# B&R Automation Studio project 8238 (part 12)

#### msgBinSearchHelpTxtLine.st
```iecst
(********************************************************************
 * COPYRIGHT -- Herbert Kannegiesser GmbH
 ********************************************************************
 * Library: KGlibMsg
 * File: msgBinSearchTxtLine.st
 * Author: kuehne
 * Created: November 29, 2011
 ********************************************************************
 * Implementation of library KGlibMsg
 ********************************************************************)

(* TODO: Add your comment here *)
FUNCTION_BLOCK msgBinSearchHelpTxtLine
	wStatus := MNMSG_STAT_NOTFOUND;
	wMsgPos := 65535;
	IF bTupel = 0 OR bTupel > 3 THEN
		RETURN;
	END_IF;
	IF bTupel = 1 THEN
		IF (wFunctionID < 1) OR (wCntMsgHelpTxt < 1) THEN
			RETURN;
		END_IF;
	END_IF;
	IF bTupel = 2 OR bTupel = 3 THEN
		IF (wFunctionID < 1) OR (wNumber < 1) OR (wCntMsgHelpTxt < 1) THEN
			RETURN;
		END_IF;
	END_IF;
	wPosMin := 0;
	wPosBeg := wPosMin;
	wPosEnd := wPosMin + wCntMsgHelpTxt - 1;
	IF wPosEnd = wPosBeg THEN
		CASE bTupel OF
			1:
				IF (MsgHelpTxtList[wPosBeg].wFunctionID = wFunctionID) THEN
					wMsgPos := wPosBeg;
					wStatus := ERR_OK;
					RETURN;
				ELSE
					RETURN;
				END_IF;
			2:
				IF (MsgHelpTxtList[wPosBeg].wFunctionID = wFunctionID) AND (MsgHelpTxtList[wPosBeg].wNumber = wNumber) THEN
					wMsgPos := wPosBeg;
					wStatus := ERR_OK;
					RETURN;
				ELSE
					RETURN;
				END_IF;
			3:
				IF (MsgHelpTxtList[wPosBeg].wFunctionID = wFunctionID) AND (MsgHelpTxtList[wPosBeg].wNumber = wNumber) AND ((MsgHelpTxtList[wPosBeg].wInstance = wInstance) OR (wInstance = 0)) THEN
					wMsgPos := wPosBeg;
					wStatus := ERR_OK;
					RETURN;
				ELSE
					RETURN;
				END_IF;
		END_CASE;
	END_IF;
	wPosMin := 1;
	wPosBeg := wPosMin;
	wPosMax := wPosMin + wCntMsgHelpTxt - 1;
	wPosEnd := wPosMin + wCntMsgHelpTxt - 1;
	wPos := (wPosMin + wPosMax) / 2;
	xPosFound := FALSE;
	WHILE NOT xPosFound DO
		IF ((wPos = (wPosBeg + 1)) OR (wPos = wPosBeg)) AND NOT xPosFound THEN
			wPos := wPosBeg;
			IF (MsgHelpTxtList[wPos].wFunctionID > wFunctionID) AND (MsgHelpTxtList[wPos + 1].wFunctionID > wFunctionID) THEN
				wPos := wPosBeg + 0;
				xPosFound := TRUE;
			ELSIF (MsgHelpTxtList[wPos].wFunctionID < wFunctionID) AND (MsgHelpTxtList[wPos + 1].wFunctionID > wFunctionID) THEN
				wPos := wPosBeg + 1;
				xPosFound := TRUE;
			ELSIF (MsgHelpTxtList[wPos].wFunctionID < wFunctionID) AND (MsgHelpTxtList[wPos + 1].wFunctionID = wFunctionID) THEN
				wPos := wPosBeg + 1;
				xPosFound := TRUE;
			ELSIF (MsgHelpTxtList[wPos].wFunctionID < wFunctionID) AND (MsgHelpTxtList[wPos + 1].wFunctionID < wFunctionID) THEN
				IF wPosEnd = (wPosBeg + 1) THEN
					wCnt := wPosBeg;
					WHILE MsgHelpTxtList[wCnt].wFunctionID < wFunctionID AND (wCnt < wPosEnd) DO
						wCnt := wCnt + 1;
					END_WHILE;
					wPos := wCnt;
				ELSE
					wPos := wPosBeg + 2;
					IF NOT (MsgHelpTxtList[wPos].wFunctionID = wFunctionID) THEN
						wCnt := wPosBeg;
						WHILE MsgHelpTxtList[wCnt].wFunctionID < wFunctionID AND (wCnt < wPosEnd) DO
							wCnt := wCnt + 1;
						END_WHILE;
						wPos := wCnt;
					END_IF;
				END_IF;
				xPosFound := TRUE;
			ELSIF (MsgHelpTxtList[wPos].wFunctionID = wFunctionID) AND (MsgHelpTxtList[wPos + 1].wFunctionID > wFunctionID) THEN
				wPos := wPosBeg + 0;
				xPosFound := TRUE;
			ELSIF (MsgHelpTxtList[wPos].wFunctionID = wFunctionID) AND (MsgHelpTxtList[wPos + 1].wFunctionID = wFunctionID) THEN
				wPos := wPosBeg + 0;
				xPosFound := TRUE;
			ELSE
				// to be sure: implement a simple algorithm with linear time here to avoid unlimited repetition
				wCnt := wPosBeg;
				WHILE MsgHelpTxtList[wCnt].wFunctionID < wFunctionID AND (wCnt < wPosEnd) DO
					wCnt := wCnt + 1;
				END_WHILE;
				wPos := wCnt;
				xPosFound := TRUE;
			END_IF;
		END_IF;
		IF ((wPos = (wPosEnd - 1)) OR (wPos = wPosEnd)) AND NOT xPosFound THEN
			wPos := wPosEnd;
			IF (MsgHelpTxtList[wPos].wFunctionID < wFunctionID) AND (MsgHelpTxtList[wPos - 1].wFunctionID < wFunctionID) THEN
				wPos := wPosEnd;
				xPosFound := TRUE;
			ELSIF (MsgHelpTxtList[wPos].wFunctionID > wFunctionID) AND (MsgHelpTxtList[wPos - 1].wFunctionID < wFunctionID) THEN
				wPos := wPosEnd - 0;
				xPosFound := TRUE;
			ELSIF (MsgHelpTxtList[wPos].wFunctionID > wFunctionID) AND (MsgHelpTxtList[wPos - 1].wFunctionID = wFunctionID) THEN
				wPos := wPosEnd - 1;
				xPosFound := TRUE;
			(* ELSIF (MsgHelpTxtList[wPos].wFunctionID > wFunctionID) AND (MsgHelpTxtList[wPos - 1].wFunctionID > wFunctionID) THEN
				wPos := wPosEnd - 1;
				xPosFound := TRUE; *)
			ELSIF (MsgHelpTxtList[wPos].wFunctionID = wFunctionID) AND (MsgHelpTxtList[wPos - 1].wFunctionID < wFunctionID) THEN
				wPos := wPosEnd - 0;
				xPosFound := TRUE;
			ELSIF (MsgHelpTxtList[wPos].wFunctionID = wFunctionID) AND (MsgHelpTxtList[wPos - 1].wFunctionID = wFunctionID) THEN
				wPos := wPosEnd - 1;
				xPosFound := TRUE;
			ELSE
				// to be sure: implement a simple algorithm with linear time here to avoid unlimited repetition
				wCnt := wPosBeg;
				WHILE MsgHelpTxtList[wCnt].wFunctionID < wFunctionID AND (wCnt < wPosEnd) DO
					wCnt := wCnt + 1;
				END_WHILE;
				wPos := wCnt;
				xPosFound := TRUE;
			END_IF;
		END_IF;
		IF NOT xPosFound THEN
			IF (MsgHelpTxtList[wPos].wFunctionID > wFunctionID) AND (MsgHelpTxtList[wPos + 1].wFunctionID > wFunctionID) THEN
				wPosMax := wPos;
				wPos := (wPosMin + wPosMax) / 2;
				IF (wPosMax - wPos) = 0 THEN
					wCnt := wPosBeg;
					WHILE MsgHelpTxtList[wCnt].wFunctionID < wFunctionID AND (wCnt < wPosEnd) DO
						wCnt := wCnt + 1;
					END_WHILE;
					wPos := wCnt;
					xPosFound := TRUE;
				END_IF;
			ELSIF (MsgHelpTxtList[wPos].wFunctionID < wFunctionID) AND (MsgHelpTxtList[wPos + 1].wFunctionID < wFunctionID) THEN
				wPosMin := wPos;
				wPos := (wPosMin + wPosMax) / 2;
				IF (wPos - wPosMin) = 0 THEN
					wCnt := wPosBeg;
					WHILE MsgHelpTxtList[wCnt].wFunctionID < wFunctionID AND (wCnt < wPosEnd) DO
						wCnt := wCnt + 1;
					END_WHILE;
					wPos := wCnt;
					xPosFound := TRUE;
				END_IF;
			ELSIF (MsgHelpTxtList[wPos].wFunctionID < wFunctionID) AND (MsgHelpTxtList[wPos + 1].wFunctionID > wFunctionID) THEN
				xPosFound := TRUE;
				wPos := wPos + 1;
			ELSIF (MsgHelpTxtList[wPos].wFunctionID < wFunctionID) AND (MsgHelpTxtList[wPos + 1].wFunctionID = wFunctionID) THEN
				xPosFound := TRUE;
				wPos := wPos + 1;
			ELSIF (MsgHelpTxtList[wPos].wFunctionID = wFunctionID) AND (MsgHelpTxtList[wPos + 1].wFunctionID > wFunctionID) THEN
				xPosFound := TRUE;
				wPos := wPos;
			ELSIF (MsgHelpTxtList[wPos].wFunctionID = wFunctionID) AND (MsgHelpTxtList[wPos + 1].wFunctionID = wFunctionID) THEN
				xPosFound := TRUE;
				wPos := wPos;
			ELSE
				// to be sure: implement a simple algorithm with linear time here to avoid unlimited repetition
				wCnt := wPosBeg;
				WHILE MsgHelpTxtList[wCnt].wFunctionID < wFunctionID AND (wCnt < wPosEnd) DO
					wCnt := wCnt + 1;
				END_WHILE;
				wPos := wCnt;
				xPosFound := TRUE;
			END_IF;
		END_IF;
	END_WHILE;
	IF MsgHelpTxtList[wPos].wFunctionID <> wFunctionID THEN
		wPosMin := wPosBeg;
		wPosMax := wPosEnd;
		wCnt := wPosBeg;
		WHILE MsgHelpTxtList[wCnt].wFunctionID <> wFunctionID AND (wCnt < wPosEnd) DO
			wCnt := wCnt + 1;
		END_WHILE;
		wPos := wCnt;
		xPosFound := TRUE;
	END_IF;
	IF bTupel = 1 THEN
		IF MsgHelpTxtList[wPos].wFunctionID = wFunctionID THEN
			wMsgPos := wPos;
			wStatus := ERR_OK;
			RETURN;
		ELSE
			RETURN;
		END_IF;
	END_IF;
	IF MsgHelpTxtList[wPos].wFunctionID = wFunctionID THEN
		//###DK2011Dec07
		wPosMinLeft := wPosMin;
		wPosMaxLeft := wPos;
		wPosBegLeft := (wPosMinLeft + wPosMaxLeft) / 2;
		xPosFoundLeft := FALSE;
		xRepeat := TRUE;
		WHILE (NOT xPosFoundLeft) AND xRepeat DO
			IF ((wPosBegLeft = (wPosBeg + 1)) OR (wPosBegLeft = wPosBeg)) AND (NOT xPosFoundLeft) AND xRepeat THEN
				wPosBegLeft := wPosBeg;
				IF (MsgHelpTxtList[wPosBegLeft].wFunctionID = wFunctionID) AND (MsgHelpTxtList[wPosBegLeft + 1].wFunctionID = wFunctionID) THEN
					xPosFoundLeft := TRUE;
					xRepeat := FALSE;
				ELSIF (MsgHelpTxtList[wPosBegLeft].wFunctionID < wFunctionID) AND (MsgHelpTxtList[wPosBegLeft + 1].wFunctionID = wFunctionID) THEN
					wPosBegLeft := wPosBeg + 1;
					xPosFoundLeft := TRUE;
					xRepeat := FALSE;
				ELSE
					xPosFoundLeft := FALSE;
					xRepeat := FALSE;
				END_IF;
			END_IF;
			IF (NOT xPosFoundLeft) AND xRepeat THEN
				IF (MsgHelpTxtList[wPosBegLeft].wFunctionID = wFunctionID) AND (MsgHelpTxtList[wPosBegLeft - 1].wFunctionID = wFunctionID) THEN
					wPosMaxLeft := wPosBegLeft;
					wPosBegLeft := (wPosMinLeft + wPosMaxLeft) / 2;
					IF (wPosMaxLeft - wPosBegLeft) = 0 THEN
						xPosFoundLeft := FALSE;
						xRepeat := FALSE;
					END_IF;
				ELSIF (MsgHelpTxtList[wPosBegLeft].wFunctionID < wFunctionID) AND (MsgHelpTxtList[wPosBegLeft - 1].wFunctionID < wFunctionID) THEN
					wPosMinLeft := wPosBegLeft;
					wPosBegLeft := (wPosMinLeft + wPosMaxLeft) / 2;
					IF (wPosMinLeft - wPosBegLeft) = 0 THEN
						xPosFoundLeft := FALSE;
						xRepeat := FALSE;
					END_IF;
				ELSIF (MsgHelpTxtList[wPosBegLeft].wFunctionID = wFunctionID) AND (MsgHelpTxtList[wPosBegLeft - 1].wFunctionID < wFunctionID) THEN
					xPosFoundLeft := TRUE;
					xRepeat := FALSE;
				ELSE
					xPosFoundLeft := FALSE;
					xRepeat := FALSE;
				END_IF;
			END_IF;
		END_WHILE;
		//###DK2011Dec07
		//###DK2011Dec07
		wPosMinRight := wPos;
		wPosMaxRight := wPosMax;
		wPosEndRight := (wPosMinRight + wPosMaxRight) / 2;
		xPosFoundRight := FALSE;
		xRepeat := TRUE;
		WHILE (NOT xPosFoundRight) AND xRepeat DO
			IF ((wPosEndRight = (wPosEnd - 1)) OR (wPosEndRight = wPosEnd)) AND (NOT xPosFoundRight) AND xRepeat THEN
				wPosEndRight := wPosEnd;
				IF (MsgHelpTxtList[wPosEndRight].wFunctionID = wFunctionID) AND (MsgHelpTxtList[wPosEndRight - 1].wFunctionID = wFunctionID) THEN
					xPosFoundRight := TRUE;
					xRepeat := FALSE;
				ELSIF (MsgHelpTxtList[wPosEndRight].wFunctionID > wFunctionID) AND (MsgHelpTxtList[wPosEndRight - 1].wFunctionID = wFunctionID) THEN
					wPosEndRight := wPosEnd - 1;
					xPosFoundRight := TRUE;
					xRepeat := FALSE;
				ELSE
					xPosFoundRight := FALSE;
					xRepeat := FALSE;
				END_IF;
			END_IF;
			IF (NOT xPosFoundRight) AND xRepeat THEN
				IF (MsgHelpTxtList[wPosEndRight].wFunctionID = wFunctionID) AND (MsgHelpTxtList[wPosEndRight + 1].wFunctionID = wFunctionID) THEN
					wPosMinRight := wPosEndRight;
					wPosEndRight := (wPosMinRight + wPosMaxRight) / 2;
					IF (wPosMinRight - wPosEndRight) = 0 THEN
						xPosFoundRight := FALSE;
						xRepeat := FALSE;
					END_IF;
				ELSIF (MsgHelpTxtList[wPosEndRight].wFunctionID > wFunctionID) AND (MsgHelpTxtList[wPosEndRight + 1].wFunctionID > wFunctionID) THEN
					wPosMaxRight := wPosEndRight;
					wPosEndRight := (wPosMinRight + wPosMaxRight) / 2;
					IF (wPosMaxRight - wPosEndRight) = 0 THEN
						xPosFoundRight := FALSE;
						xRepeat := FALSE;
					END_IF;
				ELSIF (MsgHelpTxtList[wPosEndRight].wFunctionID = wFunctionID) AND (MsgHelpTxtList[wPosEndRight + 1].wFunctionID > wFunctionID) THEN
					xPosFoundRight := TRUE;
					xRepeat := FALSE;
				ELSE
					xPosFoundRight := FALSE;
					xRepeat := FALSE;
				END_IF;
			END_IF;
		END_WHILE;
		//###DK2011Dec07
		IF NOT xPosFoundLeft THEN
			wPosBeg := wPos;
			IF (wPosBeg - 1) >= wPosMin THEN
				IF MsgHelpTxtList[wPosBeg - 1].wFunctionID = wFunctionID THEN
					wPosBeg := wPosBeg - 1;
					xRepeat := TRUE;
				ELSE
					xRepeat := FALSE;
				END_IF;
			ELSE
				xRepeat := FALSE;
			END_IF;
			WHILE xRepeat DO
				IF (wPosBeg - 1) >= wPosMin THEN
					IF MsgHelpTxtList[wPosBeg - 1].wFunctionID = wFunctionID THEN
						wPosBeg := wPosBeg - 1;
						xRepeat := TRUE;
					ELSE
						xRepeat := FALSE;
					END_IF;
				ELSE
					xRepeat := FALSE;
				END_IF;
			END_WHILE;
		ELSE
			wPosBeg := wPosBegLeft;
		END_IF;
		IF NOT xPosFoundRight THEN
			wPosEnd := wPos;
			IF (wPosEnd + 1) <= (wPosMin + wCntMsgHelpTxt - 1) THEN
				IF MsgHelpTxtList[wPosEnd + 1].wFunctionID = wFunctionID THEN
					wPosEnd := wPosEnd + 1;
					xRepeat := TRUE;
				ELSE
					xRepeat := FALSE;
				END_IF;
			ELSE
				xRepeat := FALSE;
			END_IF;
			WHILE xRepeat DO
				IF (wPosEnd + 1) <= (wPosMin + wCntMsgHelpTxt - 1) THEN
					IF MsgHelpTxtList[wPosEnd + 1].wFunctionID = wFunctionID THEN
						wPosEnd := wPosEnd + 1;
						xRepeat := TRUE;
					ELSE
						xRepeat := FALSE;
					END_IF;
				ELSE
					xRepeat := FALSE;
				END_IF;
			END_WHILE;
		ELSE
			wPosEnd := wPosEndRight;
		END_IF;
	ELSE
		RETURN;
	END_IF;
	wPosMin := wPosBeg;
	wPosMax := wPosEnd;
	wPos := (wPosMin + wPosMax) / 2;
	xPosFound := FALSE;
	IF wPosMax = wPosBeg THEN
		wPos := wPosBeg;
		xPosFound := TRUE;
	END_IF;
	WHILE NOT xPosFound DO
		IF ((wPos = (wPosBeg + 1)) OR (wPos = wPosBeg)) AND NOT xPosFound THEN
			wPos := wPosBeg;
			IF (MsgHelpTxtList[wPos].wNumber > wNumber) AND (MsgHelpTxtList[wPos + 1].wNumber > wNumber) THEN
				wPos := wPosBeg + 0;
				xPosFound := TRUE;
			ELSIF (MsgHelpTxtList[wPos].wNumber < wNumber) AND (MsgHelpTxtList[wPos + 1].wNumber > wNumber) THEN
				wPos := wPosBeg + 1;
				xPosFound := TRUE;
			ELSIF (MsgHelpTxtList[wPos].wNumber < wNumber) AND (MsgHelpTxtList[wPos + 1].wNumber = wNumber) THEN
				wPos := wPosBeg + 1;
				xPosFound := TRUE;
			ELSIF (MsgHelpTxtList[wPos].wNumber < wNumber) AND (MsgHelpTxtList[wPos + 1].wNumber < wNumber) THEN
				IF wPosEnd = (wPosBeg + 1) THEN
					wCnt := wPosBeg;
					WHILE MsgHelpTxtList[wCnt].wNumber < wNumber AND (wCnt < wPosEnd) DO
						wCnt := wCnt + 1;
					END_WHILE;
					wPos := wCnt;
				ELSE
					wPos := wPosBeg + 2;
					IF NOT (MsgHelpTxtList[wPos].wNumber = wNumber) THEN
						wCnt := wPosBeg;
						WHILE MsgHelpTxtList[wCnt].wNumber < wNumber AND (wCnt < wPosEnd) DO
							wCnt := wCnt + 1;
						END_WHILE;
						wPos := wCnt;
					END_IF;
				END_IF;
				xPosFound := TRUE;
			ELSIF (MsgHelpTxtList[wPos].wNumber = wNumber) AND (MsgHelpTxtList[wPos + 1].wNumber > wNumber) THEN
				wPos := wPosBeg + 0;
				xPosFound := TRUE;
			ELSIF (MsgHelpTxtList[wPos].wNumber = wNumber) AND (MsgHelpTxtList[wPos + 1].wNumber = wNumber) THEN
				wPos := wPosBeg + 0;
				xPosFound := TRUE;
			ELSE
				// to be sure: implement a simple algorithm with linear time here to avoid unlimited repetition
				wCnt := wPosBeg;
				WHILE MsgHelpTxtList[wCnt].wNumber < wNumber AND (wCnt < wPosEnd) DO
					wCnt := wCnt + 1;
				END_WHILE;
				wPos := wCnt;
				xPosFound := TRUE;
			END_IF;
		END_IF;
		IF ((wPos = (wPosEnd - 1)) OR (wPos = wPosEnd)) AND NOT xPosFound THEN
			wPos := wPosEnd;
			IF (MsgHelpTxtList[wPos].wNumber < wNumber) AND (MsgHelpTxtList[wPos - 1].wNumber < wNumber) THEN
				wPos := wPosEnd;
				xPosFound := TRUE;
			ELSIF (MsgHelpTxtList[wPos].wNumber > wNumber) AND (MsgHelpTxtList[wPos - 1].wNumber < wNumber) THEN
				wPos := wPosEnd - 0;
				xPosFound := TRUE;
			ELSIF (MsgHelpTxtList[wPos].wNumber > wNumber) AND (MsgHelpTxtList[wPos - 1].wNumber = wNumber) THEN
				wPos := wPosEnd - 1;
				xPosFound := TRUE;
			(* ELSIF (MsgHelpTxtList[wPos].wNumber > wNumber) AND (MsgHelpTxtList[wPos - 1].wNumber > wNumber) THEN
				wPos := wPosEnd - 1;
				xPosFound := TRUE; *)
			ELSIF (MsgHelpTxtList[wPos].wNumber = wNumber) AND (MsgHelpTxtList[wPos - 1].wNumber < wNumber) THEN
				wPos := wPosEnd - 0;
				xPosFound := TRUE;
			ELSIF (MsgHelpTxtList[wPos].wNumber = wNumber) AND (MsgHelpTxtList[wPos - 1].wNumber = wNumber) THEN
				wPos := wPosEnd - 1;
				xPosFound := TRUE;
			ELSE
				// to be sure: implement a simple algorithm with linear time here to avoid unlimited repetition
				wCnt := wPosBeg;
				WHILE MsgHelpTxtList[wCnt].wNumber < wNumber AND (wCnt < wPosEnd) DO
					wCnt := wCnt + 1;
				END_WHILE;
				wPos := wCnt;
				xPosFound := TRUE;
			END_IF;
		END_IF;
		IF NOT xPosFound THEN
			IF (MsgHelpTxtList[wPos].wNumber > wNumber) AND (MsgHelpTxtList[wPos + 1].wNumber > wNumber) THEN
				wPosMax := wPos;
				wPos := (wPosMin + wPosMax) / 2;
				IF (wPosMax - wPos) = 0 THEN
					wCnt := wPosBeg;
					WHILE MsgHelpTxtList[wCnt].wNumber < wNumber AND (wCnt < wPosEnd) DO
						wCnt := wCnt + 1;
					END_WHILE;
					wPos := wCnt;
					xPosFound := TRUE;
				END_IF;
			ELSIF (MsgHelpTxtList[wPos].wNumber < wNumber) AND (MsgHelpTxtList[wPos + 1].wNumber < wNumber) THEN
				wPosMin := wPos;
				wPos := (wPosMin + wPosMax) / 2;
				IF (wPos - wPosMin) = 0 THEN
					wCnt := wPosBeg;
					WHILE MsgHelpTxtList[wCnt].wNumber < wNumber AND (wCnt < wPosEnd) DO
						wCnt := wCnt + 1;
					END_WHILE;
					wPos := wCnt;
					xPosFound := TRUE;
				END_IF;
			ELSIF (MsgHelpTxtList[wPos].wNumber < wNumber) AND (MsgHelpTxtList[wPos + 1].wNumber > wNumber) THEN
				xPosFound := TRUE;
				wPos := wPos + 1;
			ELSIF (MsgHelpTxtList[wPos].wNumber < wNumber) AND (MsgHelpTxtList[wPos + 1].wNumber = wNumber) THEN
				xPosFound := TRUE;
				wPos := wPos + 1;
			ELSIF (MsgHelpTxtList[wPos].wNumber = wNumber) AND (MsgHelpTxtList[wPos + 1].wNumber > wNumber) THEN
				xPosFound := TRUE;
				wPos := wPos;
			ELSIF (MsgHelpTxtList[wPos].wNumber = wNumber) AND (MsgHelpTxtList[wPos + 1].wNumber = wNumber) THEN
				xPosFound := TRUE;
				wPos := wPos;
			ELSE
				// to be sure: implement a simple algorithm with linear time here to avoid unlimited repetition
				wCnt := wPosBeg;
				WHILE MsgHelpTxtList[wCnt].wNumber < wNumber AND (wCnt < wPosEnd) DO
					wCnt := wCnt + 1;
				END_WHILE;
				wPos := wCnt;
				xPosFound := TRUE;
			END_IF;
		END_IF;
	END_WHILE;
	IF MsgHelpTxtList[wPos].wNumber <> wNumber THEN
		wPosMin := wPosBeg;
		wPosMax := wPosEnd;
		wCnt := wPosBeg;
		WHILE MsgHelpTxtList[wCnt].wNumber <> wNumber AND (wCnt < wPosEnd) DO
			wCnt := wCnt + 1;
		END_WHILE;
		wPos := wCnt;
		xPosFound := TRUE;
	END_IF;
	IF MsgHelpTxtList[wPos].wNumber <> wNumber THEN
		RETURN;
	END_IF;
	IF wInstance = 0 OR bTupel = 2 THEN
		wMsgPos := wPos;
		wStatus := ERR_OK;
		RETURN;
	END_IF;
	wPosBeg := wPos;
	wPosEnd := wPos;
	IF (wPosBeg - 1) >= wPosMin THEN
		IF MsgHelpTxtList[wPosBeg - 1].wNumber = wNumber THEN
			wPosBeg := wPosBeg - 1;
			xRepeat := TRUE;
		ELSE
			xRepeat := FALSE;
		END_IF;
	ELSE
		xRepeat := FALSE;
	END_IF;
	WHILE xRepeat DO
		IF (wPosBeg - 1) >= wPosMin THEN
			IF MsgHelpTxtList[wPosBeg - 1].wNumber = wNumber THEN
				wPosBeg := wPosBeg - 1;
				xRepeat := TRUE;
			ELSE
				xRepeat := FALSE;
			END_IF;
		ELSE
			xRepeat := FALSE;
		END_IF;
	END_WHILE;
	IF (wPosEnd + 1) <= wPosMax THEN
		IF MsgHelpTxtList[wPosEnd + 1].wNumber = wNumber THEN
			wPosEnd := wPosEnd + 1;
			xRepeat := TRUE;
		ELSE
			xRepeat := FALSE;
		END_IF;
	ELSE
		xRepeat := FALSE;
	END_IF;
	WHILE xRepeat DO
		IF (wPosEnd + 1) <= wPosMax THEN
			IF MsgHelpTxtList[wPosEnd + 1].wNumber = wNumber THEN
				wPosEnd := wPosEnd + 1;
				xRepeat := TRUE;
			ELSE
				xRepeat := FALSE;
			END_IF;
		ELSE
			xRepeat := FALSE;
		END_IF;
	END_WHILE;
	wCnt := wPosBeg;
	WHILE MsgHelpTxtList[wCnt].wInstance <> wInstance AND (wCnt < wPosEnd) DO
		wCnt := wCnt + 1;
	END_WHILE;
	wPos := wCnt;
	IF MsgHelpTxtList[wPos].wInstance = wInstance THEN
		wMsgPos := wPos;
		wStatus := ERR_OK;
	END_IF;
END_FUNCTION_BLOCK
```

#### msgReplSubStr.st
```iecst
(********************************************************************
 * COPYRIGHT -- Herbert Kannegiesser GmbH
 ********************************************************************
 * Library: KGlibMsg
 * File: msgReplSubStr.st
 * Author: kuehne
 * Created: January 23, 2012
 ********************************************************************
 * Implementation of library KGlibMsg
 ********************************************************************)

(* TODO: Add your comment here *)
FUNCTION_BLOCK msgReplSubStr
	wStatus := 1;
	wMatched := 0;
	xCat := FALSE;
	IF brwcslen(ADR(utfStr)) = 0 OR brwcslen(ADR(utfSubStr)) = 0 THEN
		RETURN;
	END_IF;
	lChrPosStr := 0;
	lChrPosSubStr := 0;
	WHILE lChrPosStr < brwcslen(ADR(utfStr)) DO
		utfStrFirst := "";
		brwcsncat(ADR(utfStrFirst), ADR(utfStr) + 2 * lChrPosStr, 1);
		utfStrSecond := "";
		brwcsncat(ADR(utfStrSecond), ADR(utfSubStr) + 2 * lChrPosSubStr, 1);
		IF NOT (utfStrFirst = utfStrSecond) THEN
			IF xCat THEN
				IF (brwcslen(ADR(utfStrResult)) + lChrPosSubStr < (SIZEOF(utfStrResult) / 2)) THEN
					brwcsncat(ADR(utfStrResult), ADR(utfSubStr), lChrPosSubStr);
				ELSE
					brwcsncat(ADR(utfStrResult), ADR(utfSubStr),
					UDINT_TO_UINT(brwcslen(ADR(utfSubStr)) - (brwcslen(ADR(utfStrResult)) + brwcslen(ADR(utfSubStr)) - (SIZEOF(utfStrResult) / 2 - 1))));
				END_IF;
				xCat := FALSE;
			END_IF;
			WHILE lChrPosStr < brwcslen(ADR(utfStr)) DO
				lChrPosSubStr := 0;
				utfStrFirst := "";
				brwcsncat(ADR(utfStrFirst), ADR(utfStr) + 2 * lChrPosStr, 1);
				utfStrSecond := "";
				brwcsncat(ADR(utfStrSecond), ADR(utfSubStr) + 2 * lChrPosSubStr, 1);
				IF utfStrFirst = utfStrSecond THEN
					lChrPosStr := lChrPosStr + 1;
					lChrPosSubStr := lChrPosSubStr + 1;
					xCat := TRUE;
					EXIT;
				ELSE
					brwcsncat(ADR(utfStrResult), ADR(utfStrFirst),
					UDINT_TO_UINT(brwcslen(ADR(utfStrFirst)) - (brwcslen(ADR(utfStrResult)) + brwcslen(ADR(utfStrFirst)) - (SIZEOF(utfStrResult) / 2 - 1))));
				END_IF;
				lChrPosStr := lChrPosStr + 1;
			END_WHILE;
		ELSE
			IF lChrPosSubStr = brwcslen(ADR(utfSubStr)) - 1 THEN
				wMatched := wMatched + 1;
				wStatus := ERR_OK;
				brwcsncat(ADR(utfStrResult), ADR(utfStrToReplWith),
				UDINT_TO_UINT(brwcslen(ADR(utfStrToReplWith)) - (brwcslen(ADR(utfStrResult)) + brwcslen(ADR(utfStrToReplWith)) - (SIZEOF(utfStrResult) / 2 - 1))));
				xCat := FALSE;
			ELSE
				xCat := TRUE;
			END_IF;
			IF (lChrPosStr = brwcslen(ADR(utfStr)) - 1) AND (xCat = TRUE) THEN
				brwcsncat(ADR(utfStrResult), ADR(utfSubStr), lChrPosSubStr + 1);
			END_IF;
			lChrPosStr := lChrPosStr + 1;
			lChrPosSubStr := lChrPosSubStr + 1;
		END_IF;
	END_WHILE;
END_FUNCTION_BLOCK
```

#### msgNextChrPos.st
```iecst
(********************************************************************
 * COPYRIGHT -- Herbert Kannegiesser GmbH
 ********************************************************************
 * Library: KGlibMsg
 * File: msgNextChrPos.st
 * Author: kuehne
 * Created: February 23, 2012
 ********************************************************************
 * Implementation of library KGlibMsg
 ********************************************************************)

(* TODO: Add your comment here *)
FUNCTION_BLOCK msgNextChrPos
	wStatus := 1;
	lChrPos := 0;
	_lChrPos := lStartPos;
	_lUtfLen := brwcslen(ADR(utfStr));
	WHILE _lChrPos < _lUtfLen AND wStatus = 1 DO
		_utfChr := "";
		brwcsncat(ADR(_utfChr), ADR(utfStr) + 2 * _lChrPos, 1);
		IF _utfChr = utfChr THEN
			lChrPos := _lChrPos;
			wStatus := ERR_OK;
		END_IF;
		_lChrPos := _lChrPos + 1;
	END_WHILE;
END_FUNCTION_BLOCK
```

### mnMsg-History.txt
```
1.00.0	01.07.2011	Neu
1.01.0	02.07.2011	Index für kgMsgStatus ist wählbar
1.02.0	29.07.2011	Setzten des Machinestate.xFault
1.02.1	23.08.2011	Einzelquittierung Low-und High-Word getauscht
			Hupen-Ansteuerung Faktor 1000 für Zeitbasis ergänzt

1.03.0	08.09.2011	- Mit der Compilerdirektive "-D Test" können Testmeldungen
			  erzeugt werden.
			- Fehler behoben. Es wurde kein Änderungs-Event erzeugt, wenn eine Meldungsklasse > 0 ist
			- MNMSG_IDX_KGMSGSTATTEST eingeführt, um Testmeldungen erzeugen zu können.

1.04.0	20.09.2011	- Schaut jetzt auf mnParamStatAd.xParamOK, setzt Version 0.5 von mnParam voraus
1.05.0	20.10.2011  - Umstellung auf AS 3.0.90. Entfernung der InOut-Elemente im Interface
1.06.0	20.12.2011	- Ringbuffer aus KGstandard verwenden
1.07.1	22.12.2011	- Fehler im Init-Up (Pointer für Ringbuffer) behoben
1.07.2	19.01.2012	- Seitenumschaltung für MsgHistList
1.07.3	25.01.2012	- In MsgList werden Attribute eingefügt
1.07.4	27.01.2012	- Attribute werden in alle Text-Listen eingefügt, neue bEvent Vergabe in HistList
1.07.5	17.02.2012	- RB aus KGstdLib für HistList, noch Ungenauigkeiten bei Überlauf
1.08.1	29.02.2012	- Cleaned-up code, RB can be read properly
1.09.0	01.03.2012	- Kommandokanal zum PC an den neuen Standard angepasst
					- Überflüssige Ringbuffer entfernt
					- Test entfernt
		02.03.2012	- Schnittstellen gekapselt.
					- Kommandos an IFmnMsg bereinigt. Auch für die Visu.
					- Der Test-Teil ist wieder entfallen, da das Framework einen Testadapter erhält.
1.10.0	03.03.2012	- MNMSG_RUN_VC eingeführt. Damit ist die Aufbereitung der VC-Listen abschaltbar.
					- Die Meldungsstatistik wird auf die Version der Konfiguration hin überwacht.
1.11.0	06.03.2012	- Bugfix
					- Kompatibel mit mnTest
1.11.1	07.03.2012	- Bugfix Wartungsmeldungen. Wurden nicht eingetragen
					- Hupe wird als Status ausgegeben
1.11.3	20.03.2012	- Version von Dirk Kühne
1.11.4	20.03.2012	- Gemerget
1.11.5	20.03.2012	- Bugfix Statistik löschen
					- Abhängigkeiten ergänzt
1.11.6	20.03.2012	- asBRWStr statt asWStr
1.11.7	23.03.2012	- Bugfix. Wartungsmeldung hat geflattert.
1.11.8	23.03.2012	- Zeitstempel für geänderte Meldungslisten feiner aufgelöst.
1.11.9	05.06.2012	- Trennzeichen zwischen Funktion und Instanz
1.12.0	16.07.2012 	- Bugfix: Meldungen für DFII wurden nicht korrekt gesendet. _ReadRB wurde falsch aufgerufen.
```

### CfgMsgStat.mnMsg.txt
```
;****************************
; Meldungsmanager mnMsg
;*****************************
00002, 01000, 00000, 00000;
00002, 01003, 00000, 00000;
00002, 09999, 00000, 00000;
```

### Package Logical/Standard/Kanlink/KGFramework/Pkg_mnParam - Parameter-Manager

### mnParam.typ - Package data types
```iecst
(********************************************************************
 * COPYRIGHT -- Microsoft
 ********************************************************************
 * Package: Pkg_mnParam_Test
 * File: mnParam.typ
 * Author: hunholz
 * Created: July 23, 2011
 ********************************************************************
 * Data types of package Pkg_mnParam_Test
 ********************************************************************)

TYPE
	mnParamStatAd_typ : 	STRUCT
		xParamOK : BOOL;
		xModelImported : BOOL;
		xSystemfault : BOOL;
		dtExportContent : DATE_AND_TIME;
		HeaderVersion : mnParam_HeaderVersionRow_typ;
		utfMachineNumber : WSTRING[15];
		utfMachineName : WSTRING[31];
		sPkgVersion : STRING[10];
		wCntFilesImportOK : UINT;
		wCntFilesImportFailed : UINT;
		wCntFilesImportFound : UINT;
	END_STRUCT;
END_TYPE

(*INTERFACE*)

TYPE
	mnParam_EditNumValue_typ : 	STRUCT
		rVal : ARRAY[1..MNPARAM_CNT_EDITROWS]OF REAL;
		xSave : ARRAY[1..MNPARAM_CNT_EDITROWS]OF BOOL;
		wIdx : ARRAY[1..MNPARAM_CNT_EDITROWS]OF UINT;
	END_STRUCT;
	mnParam_EditStrValue_typ : 	STRUCT
		utfVal : ARRAY[1..MNPARAM_CNT_EDITROWS]OF WSTRING[31];
		xSave : ARRAY[1..MNPARAM_CNT_EDITROWS]OF BOOL;
		wIdx : ARRAY[1..MNPARAM_CNT_EDITROWS]OF UINT;
	END_STRUCT;
	IFmnParamOutEditNumAttr_typ : 	STRUCT
		wType : UINT;
		wParIdx : UINT;
		wFunctionID : UINT;
		wParamNo : UINT;
		wArrIdx : ARRAY[1..4]OF UINT;
		bWriteAccess : USINT;
		bReadAccess : USINT;
		wUnit : UINT;
		utfParameterName : WSTRING[63];
		utfParameterHelpTxt : WSTRING[255];
		utfInstance : WSTRING[31];
		utfFunction : WSTRING[31];
		sUnit : STRING[11];
		rMin : REAL;
		rMax : REAL;
		rDefault : REAL;
		lDigits : UDINT;
	END_STRUCT;
	IFmnParamOutEditStrAttr_typ : 	STRUCT
		wType : UINT;
		wParIdx : UINT;
		wFunctionID : UINT;
		wParamNo : UINT;
		wArrIdx : ARRAY[1..4]OF UINT;
		bWriteAccess : USINT;
		bReadAccess : USINT;
		utfParameterName : WSTRING[63];
		utfParameterHelpTxt : WSTRING[255];
		utfInstance : WSTRING[31];
		utfFunction : WSTRING[31];
		utfDefault : WSTRING[31];
		wMaxLength : UINT;
	END_STRUCT;
	IFmnParamOutEdit_typ : 	STRUCT
		wStatus : UINT;
		bContainer : USINT;
		bCntNumRows : USINT;
		bCntStrRows : USINT;
		bReserve : USINT;
		wContainerInstance : UINT;
		wRowStrCntAll : UINT;
		wRowStrOffset : UINT;
		wRowNumCntAll : UINT;
		wRowNumOffset : UINT;
		lPtrEditNumValues : UDINT;
		lPtrEditStrValues : UDINT;
		AttrNum : ARRAY[1..MNPARAM_CNT_EDITROWS]OF IFmnParamOutEditNumAttr_typ;
		AttrStr : ARRAY[1..MNPARAM_CNT_EDITROWS]OF IFmnParamOutEditStrAttr_typ;
		wCntFilesImportOK : UINT;
		wCntFilesImportFailed : UINT;
		wCntFilesImportFound : UINT;
		wCntNamelist : UINT;
		wIdxContainerNamelist : UINT;
		wParIdxNamelist : UINT;
		wNameListNo : ARRAY[1..MNPARAM_CNT_NAMELIST]OF UINT;
		utfNameListName : ARRAY[1..MNPARAM_CNT_NAMELIST]OF WSTRING[39];
		wFilterFunctionID : UINT;
		utfFilterFunction : WSTRING[31];
	END_STRUCT;
	IFmnParamOut_typ : 	STRUCT
		utfMachineNumber : WSTRING[15];
		xParamOK : BOOL;
		xModelImported : BOOL;
		xSystemfault : BOOL;
		xRequestMachineNumber : BOOL := FALSE;
		HeaderVersion : mnParam_HeaderVersionRow_typ;
		Edit : IFmnParamOutEdit_typ;
	END_STRUCT;
	IFmnParamInEdit_typ : 	STRUCT
		wCommand : UINT;
		bContainer : USINT;
		bCntNumRows : USINT;
		bCntStrRows : USINT;
		bLocUnit : USINT;
		bUserLevel : USINT;
		bSelectModeNum : USINT;
		bSelectModeStr : USINT;
		diContainerInstance : DINT;
		wContainerInstanceFrom : UINT;
		wRowStrOffset : UINT;
		wRowNumOffset : UINT;
		wSelParIdxNum : ARRAY[1..MNPARAM_CNT_EDITROWS]OF UINT;
		wSelParArrIdxNum : ARRAY[1..MNPARAM_CNT_EDITROWS,1..4]OF UINT;
		wSelParIdxStr : ARRAY[1..MNPARAM_CNT_EDITROWS]OF UINT;
		wSelParArrIdxStr : ARRAY[1..MNPARAM_CNT_EDITROWS,1..4]OF UINT;
		wSelIdxContainerNamelist : UINT;
		wSelParIdxNamelist : UINT;
		wFilterFunctionID : UINT;
	END_STRUCT;
	IFmnParamIn_typ : 	STRUCT
		utfSetMachineNumber : WSTRING[15];
		xSetMachineNumber : BOOL := FALSE;
		Edit : IFmnParamInEdit_typ;
	END_STRUCT;
	IFmnParam_typ : 	STRUCT
		In : IFmnParamIn_typ;
		Out : IFmnParamOut_typ;
	END_STRUCT;
END_TYPE
```

### mnParam.var - Package variables
```iecst
(********************************************************************
 * COPYRIGHT -- Microsoft
 ********************************************************************
 * Package: PkgMNPARAM_Test
 * File: mnParam.var
 * Author: hunholz
 * Created: July 23, 2011
 ********************************************************************
 * Variables of package PkgMNPARAM_Test
 ********************************************************************)
(*Konstanten*)
VAR CONSTANT
	MNPARAM_FUNCTIONID : UINT := 1; (*Entsprechend Zuordnungsliste*)
	MNPARAM_PATH_PM : STRING[15] := 'PM\';
	MNPARAM_PATH_EXPORT : STRING[15] := 'PM\Export\';
	MNPARAM_PATH_IMPORT : STRING[15] := 'PM\Import\';
	MNPARAM_FILESUFF : STRING[7] := '.csv';
END_VAR
(*Kommandos*)
VAR CONSTANT
	MNPARAM_CMD_NOCOMMAND : UINT := 0;
	MNPARAM_CMD_IMPORT : UINT := 1;
	MNPARAM_CMD_DELETE : UINT := 2;
	MNPARAM_CMD_FILLEDITOR : UINT := 3;
	MNPARAM_CMD_SAVEEDITOR : UINT := 4;
	MNPARAM_CMD_CREATE_INDCONT : UINT := 5;
	MNPARAM_CMD_DELETE_INDCONT : UINT := 6;
	MNPARAM_CMD_COPY_INDCONT : UINT := 7;
	MNPARAM_CMD_BACKUP : UINT := 8;
	MNPARAM_CMD_RESTORE : UINT := 9;
	MNPARAM_CMD_FILLNAMELIST : UINT := 10;
	MNPARAM_CMD_MAX : UINT := 59999;
	MNPARAM_STAT_NOCOMMAND : UINT := 0;
	MNPARAM_STAT_FILLEDITOR_OK : UINT := 3;
	MNPARAM_STAT_SAVEEDITOR_OK : UINT := 4;
	MNPARAM_STAT_CREATE_INDCONT_OK : UINT := 5;
	MNPARAM_STAT_DELETE_INDCONT_OK : UINT := 6;
	MNPARAM_STAT_COPY_INDCONT_OK : UINT := 7;
	MNPARAM_STAT_BACKUP_OK : UINT := 8;
	MNPARAM_STAT_RESTORE_OK : UINT := 9;
	MNPARAM_STAT_FILLNAMELIST_OK : UINT := 10;
	MNPARAM_STAT_DIREMPTY : UINT := 60000;
	MNPARAM_STAT_WRONGIDX : UINT := 60001;
	MNPARAM_STAT_DELPARFAULT : UINT := 60002;
	MNPARAM_STAT_DELDEFFAULT : UINT := 60003;
	MNPARAM_STAT_NUMPARNOTFOUND : UINT := 60004;
	MNPARAM_STAT_WRITEPROTECTED : UINT := 60005;
	MNPARAM_STAT_STRPARNOTFOUND : UINT := 60006;
	MNPARAM_STAT_BINPARNOTFOUN : UINT := 60007;
	MNPARAM_STAT_DELNUMPAR : UINT := 60008;
	MNPARAM_STAT_DELSTRPAR : UINT := 60009;
	MNPARAM_STAT_DELBINPAR : UINT := 60010;
	MNPARAM_STAT_DELFILE : UINT := 60011;
	MNPARAM_STAT_IMPDIRREAD : UINT := 60020;
	MNPARAM_STAT_IMPFILENOTFND : UINT := 60021;
	MNPARAM_STAT_IMPALLOCMEM : UINT := 60022;
	MNPARAM_STAT_IMPOPENFILE : UINT := 60023;
	MNPARAM_STAT_IMPREADFILE : UINT := 60024;
	MNPARAM_STAT_IMPCNTLINES : UINT := 60025;
	MNPARAM_STAT_IMPTYPE : UINT := 60026;
	MNPARAM_STAT_IMPMACHINENO : UINT := 60027;
	MNPARAM_STAT_IMPROOT : UINT := 60028;
	MNPARAM_STAT_SYSERROR : UINT := 60029;
	MNPARAM_STAT_IMPALLOCMEMN : UINT := 60030;
	MNPARAM_STAT_IMPALLOCMEMS : UINT := 60031;
	MNPARAM_STAT_IMPREADNUM : UINT := 60032;
	MNPARAM_STAT_IMPREADSTR : UINT := 60033;
	MNPARAM_STAT_IMPREADBIN : UINT := 60034;
	MNPARAM_STAT_IMPWRITENUM : UINT := 60035;
	MNPARAM_STAT_IMPWRITESTR : UINT := 60036;
	MNPARAM_STAT_IMPWRITEBIN : UINT := 60037;
	MNPARAM_STAT_EXPALLOCMEMCSV : UINT := 60038;
	MNPARAM_STAT_CREATECSV : UINT := 60039;
	MNPARAM_STAT_OPENCSV : UINT := 60040;
	MNPARAM_STAT_WRITECSV : UINT := 60041;
	MNPARAM_STAT_CLOSECSV : UINT := 60042;
	MNPARAM_STAT_NULLPOINTER : UINT := 60043; (*Nullpointerfehler*)
	MNPARAM_STAT_EXPFREEMEM : UINT := 60044; (*Speicher für Exportdatei konnte nicht wieder frei gegeben werden*)
	MNPARAM_STAT_CONTAINER_NOT_VALID : UINT := 60045; (*Container ID ist nicht gültig*)
	MNPARAM_STAT_CONTINST_NOT_VALID : UINT := 60046; (*Containerinstanz ist nich gültig*)
	MNPARAM_STAT_CONTINST_NOT_EXIST : UINT := 60047; (*Containerinstanz existiert nicht*)
	MNPARAM_STAT_CONTINST_EMPTY : UINT := 60048; (*Container ist leer*)
	MNPARAM_STAT_FREEMEM : UINT := 60049;
	MNPARAM_STAT_DIRREAD : UINT := 60050;
	MNPARAM_STAT_NOUSBSTICK : UINT := 60051;
	MNPARAM_STAT_NOIMPORTDIR : UINT := 60052;
	MNPARAM_STAT_LINKUSB : UINT := 60053;
	MNPARAM_STAT_CREATEDIR : UINT := 60054;
	MNPARAM_STAT_COPY : UINT := 60055;
	MNPARAM_STAT_CONTINST_EXIST : UINT := 60056; (*Containerinstanz existiert bereits*)
	MNPARAM_STAT_FILENOTSUPPORTED : UINT := 60057; (*Datei kann nicht importiert werden*)
	MNPARAM_STAT_NOVERSION : UINT := 60058; (*Keine Version in der Datei*)
	MNPARAM_STAT_NO_FREE_CONTINST : UINT := 60059; (*Keine freie Containerinstanz*)
END_VAR
(*Meldungen*)
VAR CONSTANT
	MNPARAM_MSG_WARN_DELETE : UINT := 2;
	MNPARAM_MSG_WARN_IMPORT : UINT := 1;
	MNPARAM_MSG_WARN_FILLEDITOR : UINT := 3;
	MNPARAM_MSG_WARN_SAVEEDITOR : UINT := 4;
	MNPARAM_MSG_WARN_BACKUP : UINT := 5;
	MNPARAM_MSG_WARN_CREATE : UINT := 6;
	MNPARAM_MSG_WARN_COPY : UINT := 7;
	MNPARAM_MSG_WARN_IMPORTFAILED : UINT := 9;
	MNPARAM_MSG_WARN_MISSINGMNO : UINT := 10;
	MNPARAM_MSG_SYSTEMERROR : UINT := 20000;
END_VAR
(*Auswahlmodi für Parameter*)
VAR CONSTANT
	MNPARAM_SELECTMODE_LINEAR : USINT := 0;
	MNPARAM_SELECTMODE_BYIDX : USINT := 1;
	MNPARAM_SELECTMODE_LINEAR_FFUNCT : USINT := 2;
END_VAR
(*Importmodi*)
VAR CONSTANT
	MNPARAM_IMPORT_DIFFERENCE : UDINT := 0; (*Es werden nur die Daten verändert, die in der Importdatei stehen.*)
	MNPARAM_IMPORT_RESTORE : UDINT := 1; (*Vor dem Import der Daten, werden alle Daten des Containers auf Default zurückgesetzt.*)
END_VAR
(*Modi zum Prüfen der Maschinennummer im Datencontainer*)
VAR CONSTANT
	MNPARAM_CMNO_CHECK : UINT := 0; (*Datencontainer mit falscher Maschinennummer werden nicht importiert.*)
	MNPARAM_CMNO_CHECKNOT : UINT := 1; (*Datencontainer werden ohne Prüfung der Maschinennummer importiert.*)
END_VAR
(*Ungueltige Maschinennummer*)
VAR CONSTANT
	MNPARAM_INVALID_MACHINENO : WSTRING[15] := "dummy";
END_VAR
(*Interface-Variablen*)
VAR
	IFmnParam : IFmnParam_typ;
	mnParamCmd : KG_Cmd_typ;
	mnParamStat : Stat_typ;
	mnParamStatAd : mnParamStatAd_typ;
END_VAR
```

### Program Logical/Standard/Kanlink/KGFramework/Pkg_mnParam/mnParam (IEC) - Parameter Manager
